{attribute addProperty BoxType "EL3783-0000-0018"}
{attribute addProperty Id "U2_SamplesAT %I*ARRAY [0..19] OF INT32040"}
{attribute addProperty CRC "339589939"}
{attribute addProperty SizeInBites "320"}
{attribute addProperty SizeInBytes "40"}
TYPE L2_Voltage_Samples_143DBB33 :
STRUCT
	{attribute addProperty Name "U2_Samples"}
	U2_Samples AT %I* : ARRAY [0..19] OF INT;
END_STRUCT
END_TYPE

(* stored: Version 1.2.0.0, ProductVersion 3.1.4024.9
   DUT L2_Voltage_Samples_143DBB33: Id {8430ecaf-9520-4d82-ad7f-797789a83d05} *)
